// TIA Portal V17 export
// export: Created 2025-06-26T06:49:17.4951211Z, ExportSetting WithDefaults, DisplayName Totally Integrated Automation Portal, DisplayVersion V17 Update 8, DisplayName TIA Portal Openness, DisplayVersion V17 Update 8, DisplayName TIA Portal Version Control Interface, DisplayVersion V17, DisplayName STEP 7 Professional, DisplayVersion V17 Update 8, DisplayName STEP 7 Safety, DisplayVersion V17 Update 6, DisplayName WinCC Advanced, DisplayVersion V17 Update 8
FUNCTION "InitAlarmLimits" : Void   // FC6, FBD
TITLE = Alarm limits
{ S7_Optimized_Access := 'TRUE' }
AUTHOR : Heaten
VERSION : 0.1
// stored: AutoNumber true, IsIECCheckEnabled false, SetENOAutomatically false, UDAEnableTagReadback false
BEGIN

REGION Network 1 (SCL): 2018 Crankcase pressure HI
   // All alarms get .bEnabled on every restart to avoid accidental/forgotten alarm deactivation
   "DB_Alarms"."2018_HBL_PT_05_High".fLimit := "DB_CurrentSetting".Compressor.Limits.p_CrankCase_Max;
   "DB_Alarms"."2018_HBL_PT_05_High".bEnable := TRUE;
END_REGION

REGION Network 2 (SCL): 2028/2115 Oil pressure LO/LOLO
   // 2028 limit is dynamic, see FB19
   "DB_Alarms"."2028_HBL_PT_17_Low".bEnable := TRUE;

   // 2115 limit is dynamic, see FB19
   "DB_Alarms"."2115_HBL_PT_17_LowLow".bEnable := TRUE;
END_REGION

REGION Network 3 (SCL): 2058/2100 Crankcase oil sump temperature LO/HI
   // 2058 Low limit is dynamic based on crankcase condensing temperature, see FB19
   "DB_Alarms"."2058_HBL_TT_03_Low".bEnable := TRUE;

   "DB_Alarms"."2100_HBL_TT_03_High".fLimit := "DB_CurrentSetting".Fluid.Limits.T_OilTemperature_Critical;
   "DB_Alarms"."2100_HBL_TT_03_High".bEnable := TRUE;
END_REGION

REGION Network 4 (SCL): 2101 Heat sink suction temperature HI
   "DB_Alarms"."2101_HBL_TT_901_High".bEnable := TRUE;
   "DB_Alarms"."2101_HBL_TT_901_High".fLimit := "DB_CurrentSetting".MissingSetting.Misc.T_HeatSinkTemperatureIn_Max;
END_REGION

REGION Network 5 (SCL): 2102/2116 Compressor discharge pressure HI/HI HI
   // 100kPa below the HIHI limit (2116)
   // 100kPa below the HIHI limit
   "DB_Alarms"."2102_HBL_PT_503_High".fLimit := "DB_CurrentSetting".System.Limits.p_CompressorOut_Max - 100.0;
   "DB_Alarms"."2102_HBL_PT_503_High".bEnable := TRUE;

   "DB_Alarms"."2116_HBL_PT_503_HighHigh".bEnable := TRUE;
   "DB_Alarms"."2116_HBL_PT_503_HighHigh".fLimit := "DB_CurrentSetting".System.Limits.p_CompressorOut_Max;
END_REGION

REGION Network 6 (SCL): 2103 Heat sink discharge temperature HI
   "DB_Alarms"."2103_HBL_TT_518_High".fLimit := "DB_CurrentSetting".Fluid.Limits.T_HeatSinkTemperature_Max;
   "DB_Alarms"."2103_HBL_TT_518_High".bEnable := TRUE;
END_REGION

REGION Network 7 (SCL): 2105 Heat source suction temperature HI
   "DB_Alarms"."2105_HBL_TT_546_High".fLimit := "DB_CurrentSetting".Fluid.Limits.T_HeatSourceTemperature_Max;
   "DB_Alarms"."2105_HBL_TT_546_High".bEnable := TRUE;
END_REGION

REGION Network 8 (SCL): 2106 Control cabinet air temperature HI
   "DB_Alarms"."2106_HBL_TT_17_High".fLimit := "DB_CurrentSetting".StaticSetting.Limits.T_Cabinet_Max;
   "DB_Alarms"."2106_HBL_TT_17_High".bEnable := TRUE;
END_REGION

REGION Network 9 (SCL): 2107 Container air temperature HI
   "DB_Alarms"."2107_HBL_TT_16_High".fLimit := "DB_CurrentSetting".System.Limits.T_Housing_Max;
   "DB_Alarms"."2107_HBL_TT_16_High".bEnable := TRUE;
END_REGION

REGION Network 10 (SCL): 2108 Ambient air temperature HI
   "DB_Alarms"."2108_HBL_TT_18_High".fLimit := "DB_CurrentSetting".StaticSetting.Limits.T_Ambient_Max;
   "DB_Alarms"."2108_HBL_TT_18_High".bEnable := TRUE;
END_REGION

REGION Network 11 (SCL): 2109 Compressor motor temperature HI
   "DB_Alarms"."2109_HBL_TT_20_High".fLimit := "DB_CurrentSetting".Compressor.Limits.T_Motor_Max;
   "DB_Alarms"."2109_HBL_TT_20_High".bEnable := TRUE;
END_REGION

REGION Network 12 (SCL): 2110/2111 Oil sump wall temperature HI
   // Leave a temperature margin to avoid actually getting up into the critical temperature before triggering
   "DB_Alarms"."2110_HBL_TT_21_High".fLimit := "DB_CurrentSetting".Fluid.Limits.T_OilTemperature_Critical - 20.0;
   "DB_Alarms"."2110_HBL_TT_21_High".bEnable := TRUE;

   "DB_Alarms"."2111_HBL_TT_22_High".fLimit := "DB_CurrentSetting".Fluid.Limits.T_OilTemperature_Critical - 20.0;
   "DB_Alarms"."2111_HBL_TT_22_High".bEnable := TRUE;
END_REGION

REGION Network 13 (SCL): 2112 Oil separator oil level HI
   // ##FIX not in DB_CurrentSettings yet (or ever will be?)
   "DB_Alarms"."2112_HBL_LT_02_High".fLimit := 80.0;
   "DB_Alarms"."2112_HBL_LT_02_High".bEnable := TRUE;
END_REGION

REGION Network 14 (SCL): 2113/2114 Gas detectors HI
   // ##FIX not in DB_CurrentSettings yet
   "DB_Alarms"."2113_HBL_CT_01_High".fLimit := 1000.0;
   "DB_Alarms"."2113_HBL_CT_01_High".bEnable := TRUE;

   "DB_Alarms"."2114_HBL_CT_615_High".fLimit := 1000.0;
   "DB_Alarms"."2114_HBL_CT_615_High".bEnable := TRUE;
END_REGION

REGION Network 15 (SCL): 2301/2302 Heat source temperature rate of change
   // ##FIX not in DB_CurrentSettings yet
   "DB_Alarms"."2301_HeatSourceTempDropCritical".fLimit := -0.25;
   "DB_Alarms"."2301_HeatSourceTempDropCritical".bEnable := TRUE;

   "DB_Alarms"."2302_HeatSourceTempRiseCritical".fLimit := 0.25;
   "DB_Alarms"."2302_HeatSourceTempRiseCritical".bEnable := TRUE;
END_REGION

REGION Network 16 (SCL): 2303/2304 Superheat compressor suction HI/LO
   // ##FIX These limits are not in DB_CurrentSettings yet
   "DB_Alarms"."2303_SuperheatCompressor_High".fLimit := 30.0;
   "DB_Alarms"."2303_SuperheatCompressor_High".bEnable := TRUE;


   "DB_Alarms"."2304_SuperheatCompressor_Low".fLimit := "DB_CurrentSetting".System.Limits.T_SuperHeatCompressorIn_Min;
   "DB_Alarms"."2304_SuperheatCompressor_Low".bEnable := True;
END_REGION

REGION Network 17 (SCL): 2305/2306 Oil filter delta P HI/HIHI
   "DB_Alarms"."2305_OilFilterDeltaP_High".fLimit := "DB_CurrentSetting".MissingSetting.Compressor.OilFilterDeltaPWarning;
   "DB_Alarms"."2305_OilFilterDeltaP_High".bEnable := TRUE;

   "DB_Alarms"."2306_OilFilterDeltaP_HighHigh".fLimit := "DB_CurrentSetting".MissingSetting.Compressor.OilFilterDeltaPCritical;
   "DB_Alarms"."2306_OilFilterDeltaP_HighHigh".bEnable := TRUE;
END_REGION

REGION Network 18 (SCL): 2308 Evaporator discharge pressure HI
   "DB_Alarms"."2308_EvaporatorDischargePressureHigh".fLimit := "DB_CurrentSetting".System.Limits.p_EvaporatorOut_Max;
   "DB_Alarms"."2308_EvaporatorDischargePressureHigh".bEnable := TRUE;
END_REGION

REGION Network 19 (SCL): 5205 CPC tank level HI
   "DB_Alarms"."5205_CPC_LT_870_High".fLimit := 90.0;
   "DB_Alarms"."5205_CPC_LT_870_High".bEnable := TRUE;
END_REGION

REGION Network 20 (SCL): 5257 SSC barrier reservoir LO
   "DB_Alarms"."5257_SSC_LT_01_Low".fLimit := 5.0;
   "DB_Alarms"."5257_SSC_LT_01_Low".bEnable := TRUE;
END_REGION

REGION Network 21 (SCL): 5258 SSC barrier fluid pump differential pressure HI
   "DB_Alarms"."5258_SSC_PDT_01_High".fLimit := 200.0;
   "DB_Alarms"."5258_SSC_PDT_01_High".bEnable := TRUE;
END_REGION

REGION Network 22 (SCL): 5259 SSC seal discharge temperature HI
   "DB_Alarms"."5259_SSC_TT_02_High".fLimit := 110.0;
   "DB_Alarms"."5259_SSC_TT_02_High".bEnable := TRUE;
END_REGION

REGION Network 23 (SCL): 5260 SSC circulation pump suction temperature LO
   "DB_Alarms"."5260_SSC_TT_03_Low".fLimit := 10.0;
   "DB_Alarms"."5260_SSC_TT_03_Low".bEnable := TRUE;
END_REGION

REGION Network 24 (SCL): 5261/5263 SSC accumulator pressure LO/HI
   "DB_Alarms"."5261_SSC_PIT_01_Low".fLimit := 840.0;
   "DB_Alarms"."5261_SSC_PIT_01_Low".bEnable := TRUE;

   "DB_Alarms"."5263_SSC_PIT_01_High".fLimit := 1400.0;
   "DB_Alarms"."5263_SSC_PIT_01_High".bEnable := TRUE;
END_REGION

REGION Network 25 (SCL): 5262 SSC seal delta T HI
   "DB_Alarms"."5262_DeltaT_ShaftSealHigh".fLimit := 11.0;
   "DB_Alarms"."5262_DeltaT_ShaftSealHigh".bEnable := TRUE;
END_REGION
END_FUNCTION
